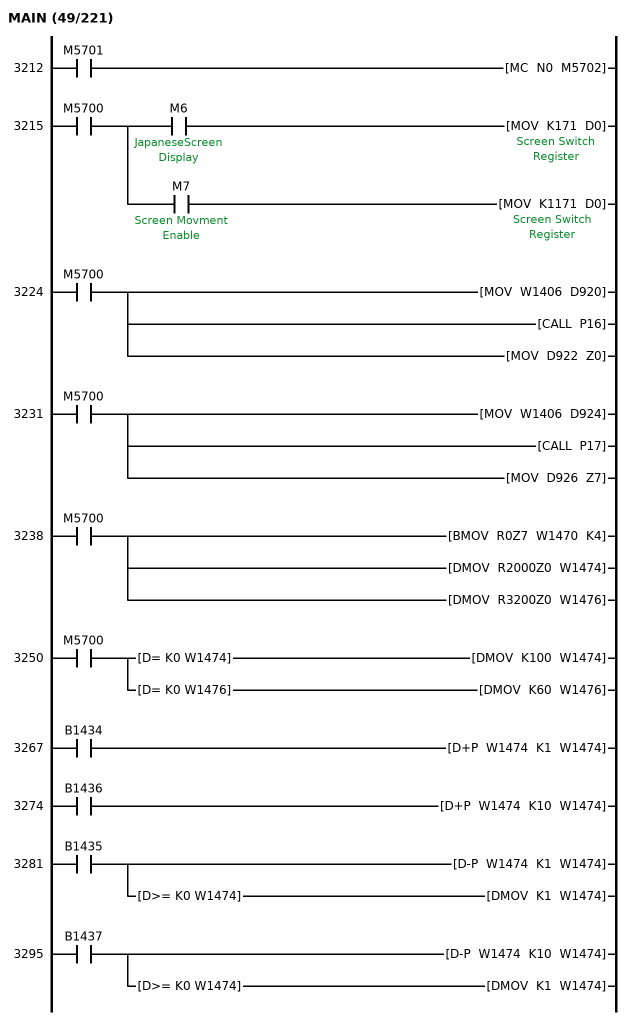
[picture p48: ladder of MAIN, rungs at steps 3212 to 3295]
3212  LD      M5701
      MC      N0 M5702
3215  LD      M5700
      MPS
      AND     M6  ; JapaneseScreen Display
      MOV     K171 D0
      MPP
      AND     M7  ; Screen Movment Enable
      MOV     K1171 D0
3224  LD      M5700
      MOV     W1406 D920
      CALL    P16
      MOV     D922 Z0
3231  LD      M5700
      MOV     W1406 D924
      CALL    P17
      MOV     D926 Z7
3238  LD      M5700
      BMOV    R0Z7 W1470 K4
      DMOV    R2000Z0 W1474
      DMOV    R3200Z0 W1476
3250  LD      M5700
      MPS
      ANDD=   K0 W1474
      DMOV    K100 W1474
      MPP
      ANDD=   K0 W1476
      DMOV    K60 W1476
3267  LD      B1434
      D+P     W1474 K1 W1474
3274  LD      B1436
      D+P     W1474 K10 W1474
3281  LD      B1435
      D-P     W1474 K1 W1474
      ANDD>=  K0 W1474
      DMOV    K1 W1474
3295  LD      B1437
      D-P     W1474 K10 W1474
      ANDD>=  K0 W1474
      DMOV    K1 W1474
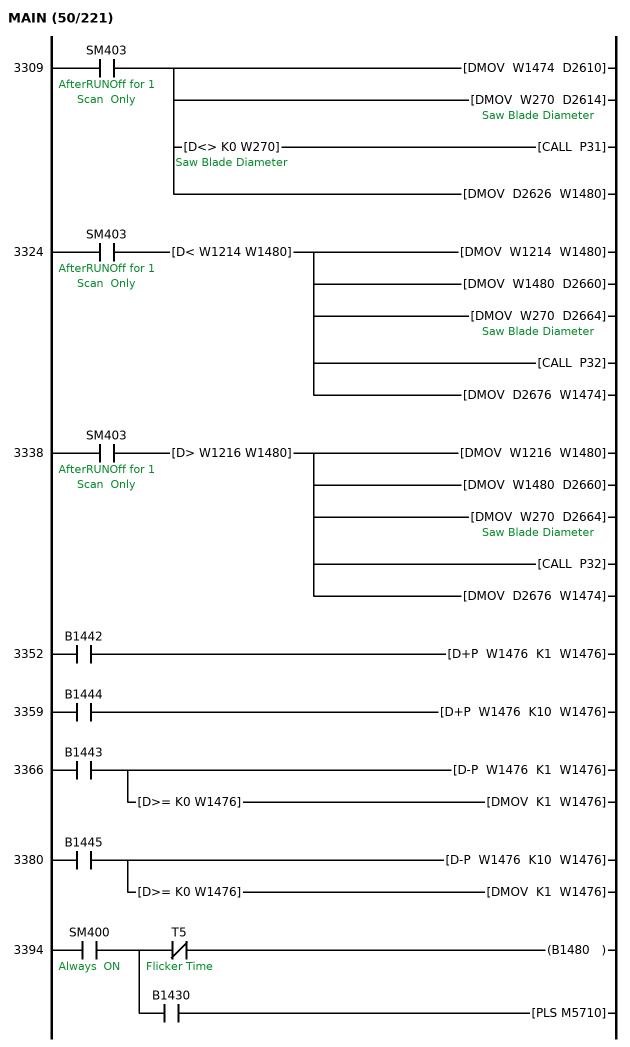
3309  LD      SM403  ; AfterRUNOff for 1 Scan  Only
      DMOV    W1474 D2610
      DMOV    W270 D2614
      MPS
      ANDD<>  K0 W270  ; Saw Blade Diameter
      CALL    P31
      MPP
      DMOV    D2626 W1480
3324  LD      SM403  ; AfterRUNOff for 1 Scan  Only
      ANDD<   W1214 W1480
      DMOV    W1214 W1480
      DMOV    W1480 D2660
      DMOV    W270 D2664
      CALL    P32
      DMOV    D2676 W1474
3338  LD      SM403  ; AfterRUNOff for 1 Scan  Only
      ANDD>   W1216 W1480
      DMOV    W1216 W1480
      DMOV    W1480 D2660
      DMOV    W270 D2664
      CALL    P32
      DMOV    D2676 W1474
3352  LD      B1442
      D+P     W1476 K1 W1476
3359  LD      B1444
      D+P     W1476 K10 W1476
3366  LD      B1443
      D-P     W1476 K1 W1476
      ANDD>=  K0 W1476
      DMOV    K1 W1476
3380  LD      B1445
      D-P     W1476 K10 W1476
      ANDD>=  K0 W1476
      DMOV    K1 W1476
3394  LD      SM400  ; Always  ON
      MPS
      ANI     T5  ; Flicker Time
      OUT     B1480
      MPP
      AND     B1430
      PLS     M5710
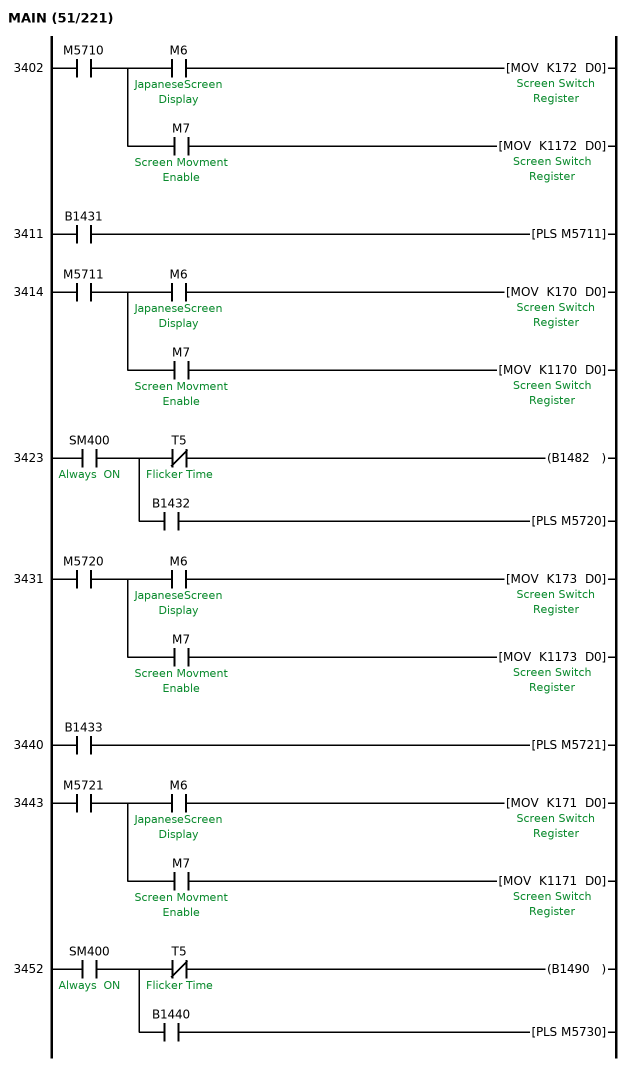
3402  LD      M5710
      MPS
      AND     M6  ; JapaneseScreen Display
      MOV     K172 D0
      MPP
      AND     M7  ; Screen Movment Enable
      MOV     K1172 D0
3411  LD      B1431
      PLS     M5711
3414  LD      M5711
      MPS
      AND     M6  ; JapaneseScreen Display
      MOV     K170 D0
      MPP
      AND     M7  ; Screen Movment Enable
      MOV     K1170 D0
3423  LD      SM400  ; Always  ON
      MPS
      ANI     T5  ; Flicker Time
      OUT     B1482
      MPP
      AND     B1432
      PLS     M5720
3431  LD      M5720
      MPS
      AND     M6  ; JapaneseScreen Display
      MOV     K173 D0
      MPP
      AND     M7  ; Screen Movment Enable
      MOV     K1173 D0
3440  LD      B1433
      PLS     M5721
3443  LD      M5721
      MPS
      AND     M6  ; JapaneseScreen Display
      MOV     K171 D0
      MPP
      AND     M7  ; Screen Movment Enable
      MOV     K1171 D0
3452  LD      SM400  ; Always  ON
      MPS
      ANI     T5  ; Flicker Time
      OUT     B1490
      MPP
      AND     B1440
      PLS     M5730
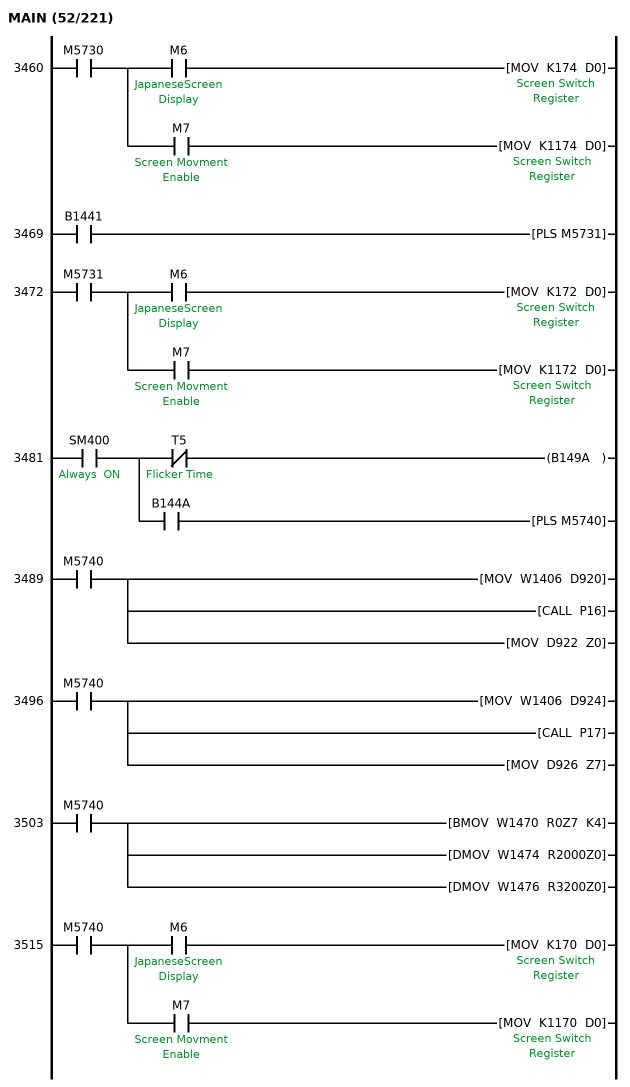
3460  LD      M5730
      MPS
      AND     M6  ; JapaneseScreen Display
      MOV     K174 D0
      MPP
      AND     M7  ; Screen Movment Enable
      MOV     K1174 D0
3469  LD      B1441
      PLS     M5731
3472  LD      M5731
      MPS
      AND     M6  ; JapaneseScreen Display
      MOV     K172 D0
      MPP
      AND     M7  ; Screen Movment Enable
      MOV     K1172 D0
3481  LD      SM400  ; Always  ON
      MPS
      ANI     T5  ; Flicker Time
      OUT     B149A
      MPP
      AND     B144A
      PLS     M5740
3489  LD      M5740
      MOV     W1406 D920
      CALL    P16
      MOV     D922 Z0
3496  LD      M5740
      MOV     W1406 D924
      CALL    P17
      MOV     D926 Z7
3503  LD      M5740
      BMOV    W1470 R0Z7 K4
      DMOV    W1474 R2000Z0
      DMOV    W1476 R3200Z0
3515  LD      M5740
      MPS
      AND     M6  ; JapaneseScreen Display
      MOV     K170 D0
      MPP
      AND     M7  ; Screen Movment Enable
      MOV     K1170 D0
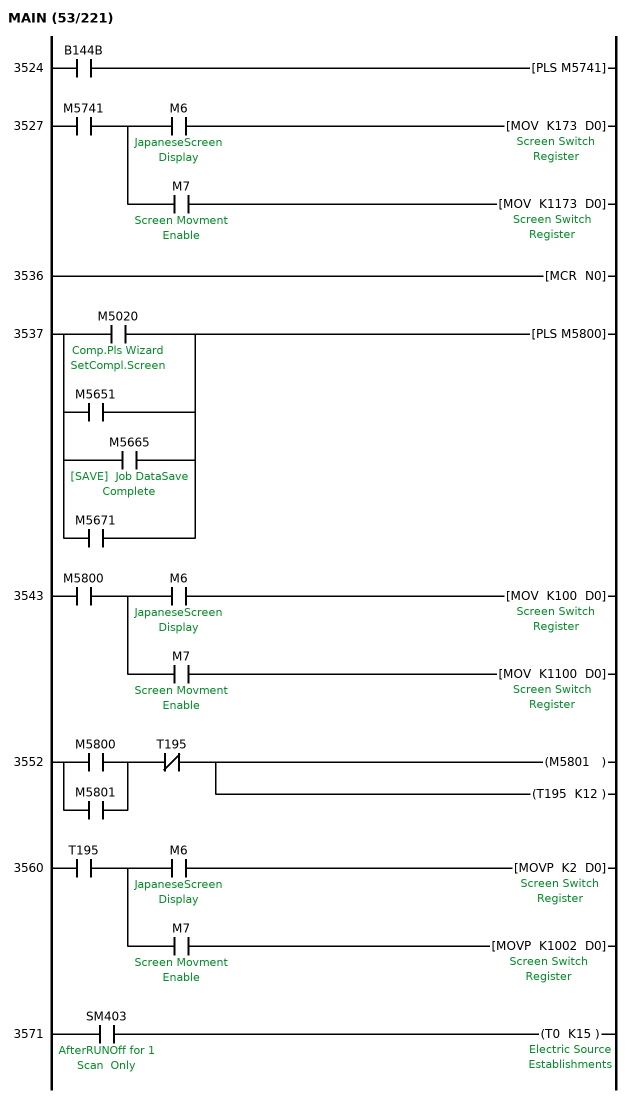
3524  LD      B144B
      PLS     M5741
3527  LD      M5741
      MPS
      AND     M6  ; JapaneseScreen Display
      MOV     K173 D0
      MPP
      AND     M7  ; Screen Movment Enable
      MOV     K1173 D0
3536  MCR     N0
3537  LD      M5020  ; Comp.Pls Wizard SetCompl.Screen
      OR      M5651
      OR      M5665  ; [SAVE]  Job DataSave Complete
      OR      M5671
      PLS     M5800
3543  LD      M5800
      MPS
      AND     M6  ; JapaneseScreen Display
      MOV     K100 D0
      MPP
      AND     M7  ; Screen Movment Enable
      MOV     K1100 D0
3552  LD      M5800
      OR      M5801
      ANI     T195
      OUT     M5801
      OUT     T195 K12
3560  LD      T195
      MPS
      AND     M6  ; JapaneseScreen Display
      MOVP    K2 D0
      MPP
      AND     M7  ; Screen Movment Enable
      MOVP    K1002 D0
3571  LD      SM403  ; AfterRUNOff for 1 Scan  Only
      OUT     T0 K15  ; Electric Source Establishments
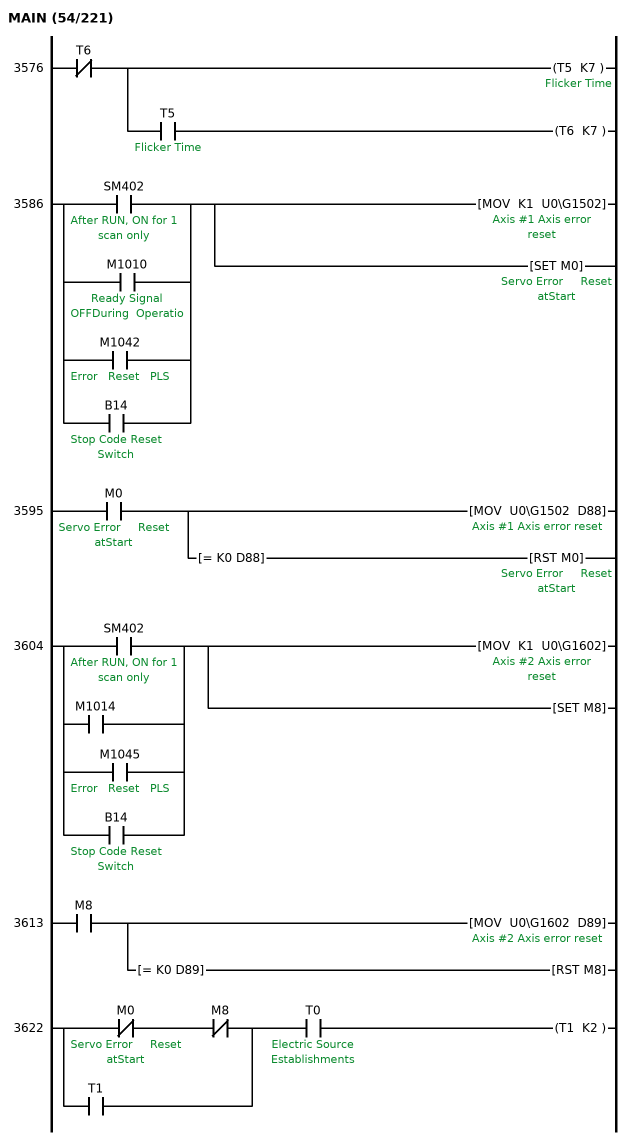
3576  LDI     T6
      OUT     T5 K7  ; Flicker Time
      AND     T5  ; Flicker Time
      OUT     T6 K7
3586  LD      SM402  ; After RUN, ON for 1 scan only
      OR      M1010  ; Ready Signal OFFDuring  Operatio
      OR      M1042  ; Error   Reset   PLS
      OR      B14  ; Stop Code Reset Switch
      MOV     K1 U0\G1502  ; Axis #1 Axis error reset
      SET     M0  ; Servo Error     Reset atStart
3595  LD      M0  ; Servo Error     Reset atStart
      MOV     U0\G1502 D88
      AND=    K0 D88
      RST     M0  ; Servo Error     Reset atStart
3604  LD      SM402  ; After RUN, ON for 1 scan only
      OR      M1014
      OR      M1045  ; Error   Reset   PLS
      OR      B14  ; Stop Code Reset Switch
      MOV     K1 U0\G1602  ; Axis #2 Axis error reset
      SET     M8
3613  LD      M8
      MOV     U0\G1602 D89
      AND=    K0 D89
      RST     M8
3622  LDI     M0  ; Servo Error     Reset atStart
      ANI     M8
      OR      T1
      AND     T0  ; Electric Source Establishments
      OUT     T1 K2
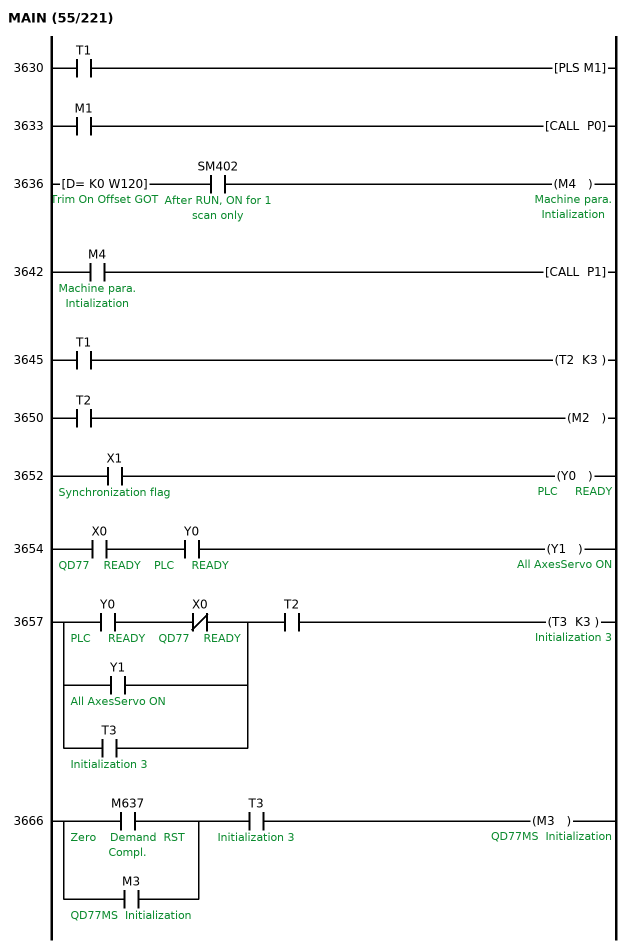
3630  LD      T1
      PLS     M1
3633  LD      M1
      CALL    P0
3636  LDD=    K0 W120  ; Trim On Offset GOT
      AND     SM402  ; After RUN, ON for 1 scan only
      OUT     M4  ; Machine para.   Intialization
3642  LD      M4  ; Machine para.   Intialization
      CALL    P1
3645  LD      T1
      OUT     T2 K3
3650  LD      T2
      OUT     M2
3652  LD      X1  ; Synchronization flag
      OUT     Y0  ; PLC     READY
3654  LD      X0  ; QD77    READY
      AND     Y0  ; PLC     READY
      OUT     Y1  ; All AxesServo ON
3657  LD      Y0  ; PLC     READY
      ANI     X0  ; QD77    READY
      OR      Y1  ; All AxesServo ON
      OR      T3  ; Initialization 3
      AND     T2
      OUT     T3 K3  ; Initialization 3
3666  LD      M637  ; Zero    Demand  RST     Compl.
      OR      M3  ; QD77MS  Initialization
      AND     T3  ; Initialization 3
      OUT     M3  ; QD77MS  Initialization
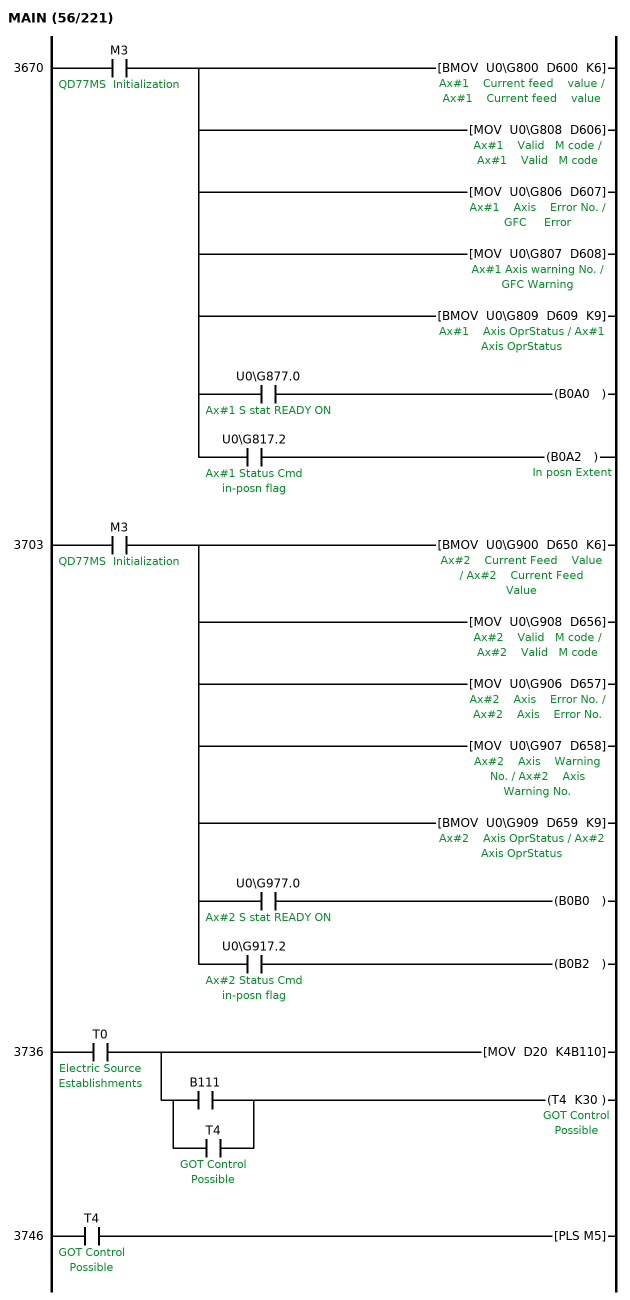
3670  LD      M3  ; QD77MS  Initialization
      BMOV    U0\G800 D600 K6  ; Ax#1    Current feed    value / Ax#1    Current feed    value
      MOV     U0\G808 D606  ; Ax#1    Valid   M code / Ax#1    Valid   M code
      MOV     U0\G806 D607  ; Ax#1    Axis    Error No. / GFC     Error
      MOV     U0\G807 D608  ; Ax#1 Axis warning No. / GFC Warning
      BMOV    U0\G809 D609 K9  ; Ax#1    Axis OprStatus / Ax#1    Axis OprStatus
      MPS
      AND     U0\G877.0  ; Ax#1 S stat READY ON
      OUT     B0A0
      MPP
      AND     U0\G817.2  ; Ax#1 Status Cmd in-posn flag
      OUT     B0A2  ; In posn Extent
3703  LD      M3  ; QD77MS  Initialization
      BMOV    U0\G900 D650 K6  ; Ax#2    Current Feed    Value / Ax#2    Current Feed    Value
      MOV     U0\G908 D656  ; Ax#2    Valid   M code / Ax#2    Valid   M code
      MOV     U0\G906 D657  ; Ax#2    Axis    Error No. / Ax#2    Axis    Error No.
      MOV     U0\G907 D658  ; Ax#2    Axis    Warning No. / Ax#2    Axis    Warning No.
      BMOV    U0\G909 D659 K9  ; Ax#2    Axis OprStatus / Ax#2    Axis OprStatus
      MPS
      AND     U0\G977.0  ; Ax#2 S stat READY ON
      OUT     B0B0
      MPP
      AND     U0\G917.2  ; Ax#2 Status Cmd in-posn flag
      OUT     B0B2
3736  LD      T0  ; Electric Source Establishments
      MOV     D20 K4B110
      LD      B111
      OR      T4  ; GOT Control     Possible
      ANB
      OUT     T4 K30  ; GOT Control     Possible
3746  LD      T4  ; GOT Control     Possible
      PLS     M5
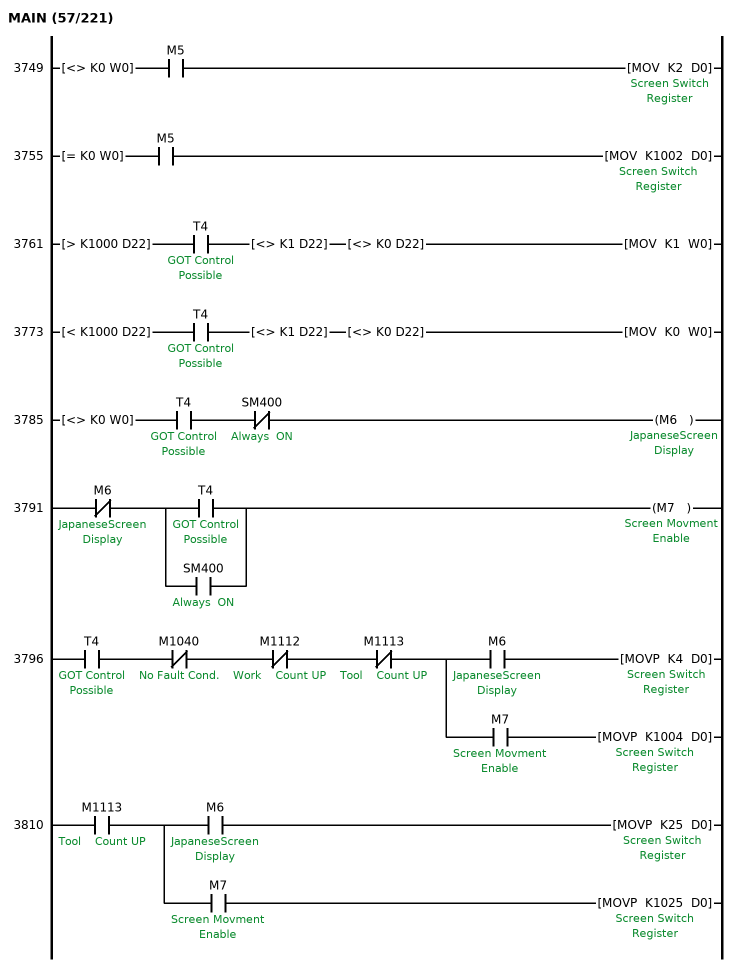
3749  LD<>    K0 W0
      AND     M5
      MOV     K2 D0
3755  LD=     K0 W0
      AND     M5
      MOV     K1002 D0
3761  LD>     K1000 D22
      AND     T4  ; GOT Control     Possible
      AND<>   K1 D22
      AND<>   K0 D22
      MOV     K1 W0
3773  LD<     K1000 D22
      AND     T4  ; GOT Control     Possible
      AND<>   K1 D22
      AND<>   K0 D22
      MOV     K0 W0
3785  LD<>    K0 W0
      AND     T4  ; GOT Control     Possible
      ANI     SM400  ; Always  ON
      OUT     M6  ; JapaneseScreen Display
3791  LDI     M6  ; JapaneseScreen Display
      LD      T4  ; GOT Control     Possible
      OR      SM400  ; Always  ON
      ANB
      OUT     M7  ; Screen Movment Enable
3796  LD      T4  ; GOT Control     Possible
      ANI     M1040  ; No Fault Cond.
      ANI     M1112  ; Work    Count UP
      ANI     M1113  ; Tool    Count UP
      MPS
      AND     M6  ; JapaneseScreen Display
      MOVP    K4 D0
      MPP
      AND     M7  ; Screen Movment Enable
      MOVP    K1004 D0
3810  LD      M1113  ; Tool    Count UP
      MPS
      AND     M6  ; JapaneseScreen Display
      MOVP    K25 D0
      MPP
      AND     M7  ; Screen Movment Enable
      MOVP    K1025 D0
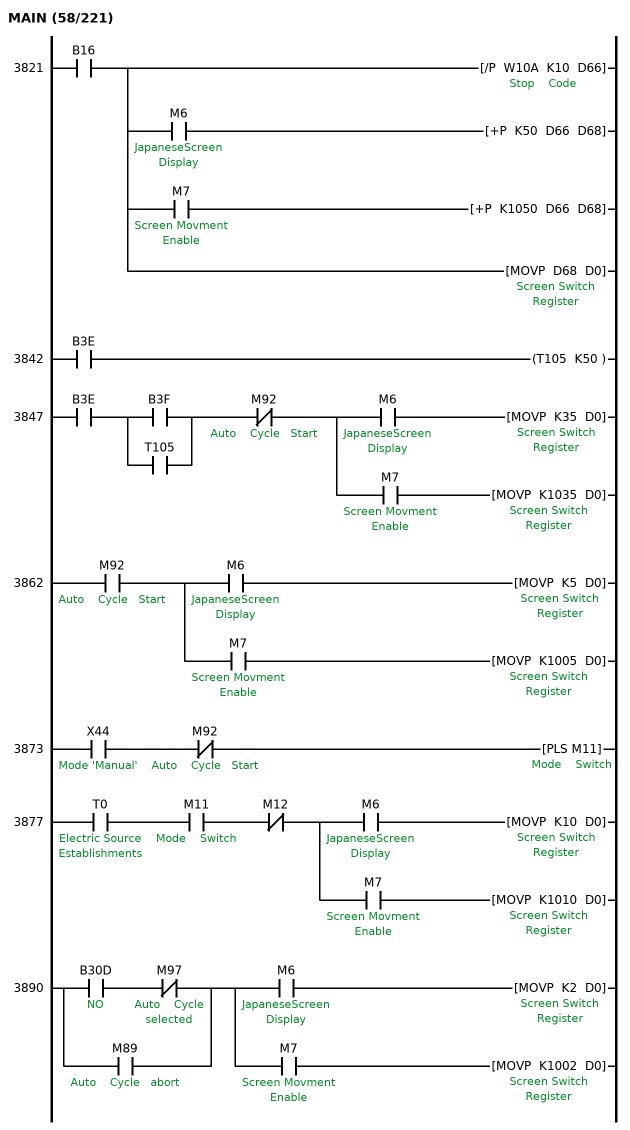
3821  LD      B16
      /P      W10A K10 D66  ; Stop    Code
      MPS
      AND     M6  ; JapaneseScreen Display
      +P      K50 D66 D68
      MRD
      AND     M7  ; Screen Movment Enable
      +P      K1050 D66 D68
      MPP
      MOVP    D68 D0
3842  LD      B3E
      OUT     T105 K50
3847  LD      B3E
      LD      B3F
      OR      T105
      ANB
      ANI     M92  ; Auto    Cycle   Start
      MPS
      AND     M6  ; JapaneseScreen Display
      MOVP    K35 D0
      MPP
      AND     M7  ; Screen Movment Enable
      MOVP    K1035 D0
3862  LD      M92  ; Auto    Cycle   Start
      MPS
      AND     M6  ; JapaneseScreen Display
      MOVP    K5 D0
      MPP
      AND     M7  ; Screen Movment Enable
      MOVP    K1005 D0
3873  LD      X44  ; Mode 'Manual'
      ANI     M92  ; Auto    Cycle   Start
      PLS     M11  ; Mode    Switch
3877  LD      T0  ; Electric Source Establishments
      AND     M11  ; Mode    Switch
      ANI     M12
      MPS
      AND     M6  ; JapaneseScreen Display
      MOVP    K10 D0
      MPP
      AND     M7  ; Screen Movment Enable
      MOVP    K1010 D0
3890  LD      B30D  ; NO
      ANI     M97  ; Auto    Cycle   selected
      OR      M89  ; Auto    Cycle   abort
      MPS
      AND     M6  ; JapaneseScreen Display
      MOVP    K2 D0
      MPP
      AND     M7  ; Screen Movment Enable
      MOVP    K1002 D0
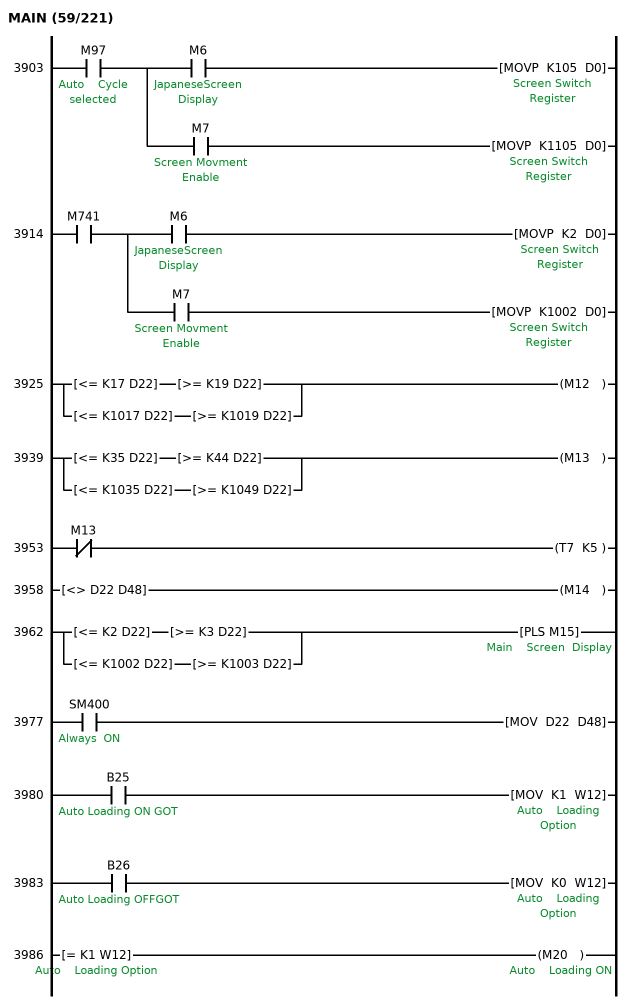
3903  LD      M97  ; Auto    Cycle   selected
      MPS
      AND     M6  ; JapaneseScreen Display
      MOVP    K105 D0
      MPP
      AND     M7  ; Screen Movment Enable
      MOVP    K1105 D0
3914  LD      M741
      MPS
      AND     M6  ; JapaneseScreen Display
      MOVP    K2 D0
      MPP
      AND     M7  ; Screen Movment Enable
      MOVP    K1002 D0
3925  LD<=    K17 D22
      AND>=   K19 D22
      LD<=    K1017 D22
      AND>=   K1019 D22
      ORB
      OUT     M12
3939  LD<=    K35 D22
      AND>=   K44 D22
      LD<=    K1035 D22
      AND>=   K1049 D22
      ORB
      OUT     M13
3953  LDI     M13
      OUT     T7 K5
3958  LD<>    D22 D48
      OUT     M14
3962  LD<=    K2 D22
      AND>=   K3 D22
      LD<=    K1002 D22
      AND>=   K1003 D22
      ORB
      PLS     M15  ; Main    Screen  Display
3977  LD      SM400  ; Always  ON
      MOV     D22 D48
3980  LD      B25  ; Auto Loading ON GOT
      MOV     K1 W12  ; Auto    Loading Option
3983  LD      B26  ; Auto Loading OFFGOT
      MOV     K0 W12
3986  LD=     K1 W12  ; Auto    Loading Option
      OUT     M20  ; Auto    Loading ON
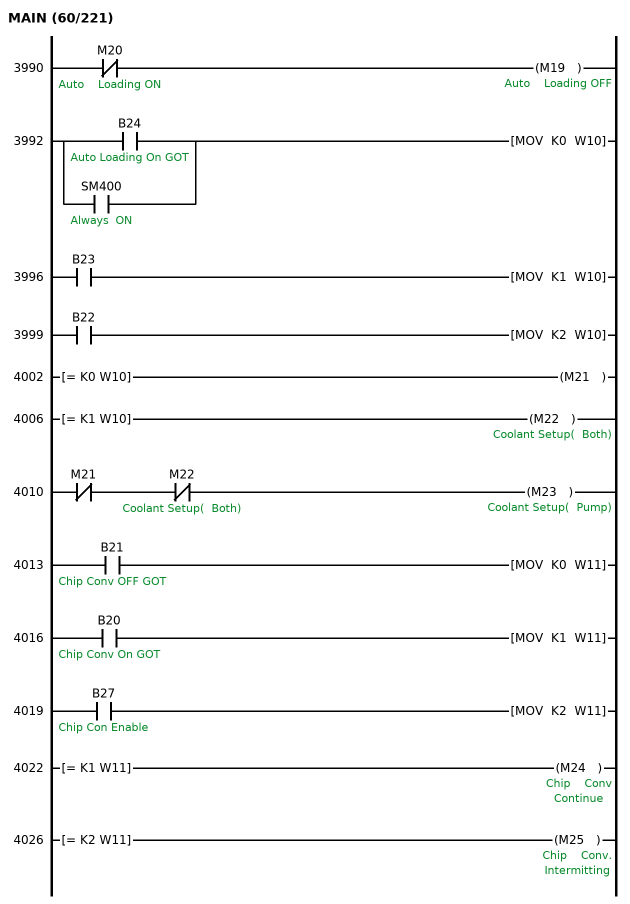
3990  LDI     M20  ; Auto    Loading ON
      OUT     M19  ; Auto    Loading OFF
3992  LD      B24  ; Auto Loading On GOT
      OR      SM400  ; Always  ON
      MOV     K0 W10
3996  LD      B23
      MOV     K1 W10
3999  LD      B22
      MOV     K2 W10
4002  LD=     K0 W10
      OUT     M21
4006  LD=     K1 W10
      OUT     M22  ; Coolant Setup(  Both)
4010  LDI     M21
      ANI     M22  ; Coolant Setup(  Both)
      OUT     M23  ; Coolant Setup(  Pump)
4013  LD      B21  ; Chip Conv OFF GOT
      MOV     K0 W11
4016  LD      B20  ; Chip Conv On GOT
      MOV     K1 W11
4019  LD      B27  ; Chip Con Enable
      MOV     K2 W11
4022  LD=     K1 W11
      OUT     M24  ; Chip    Conv    Continue
4026  LD=     K2 W11
      OUT     M25  ; Chip    Conv.   Intermitting
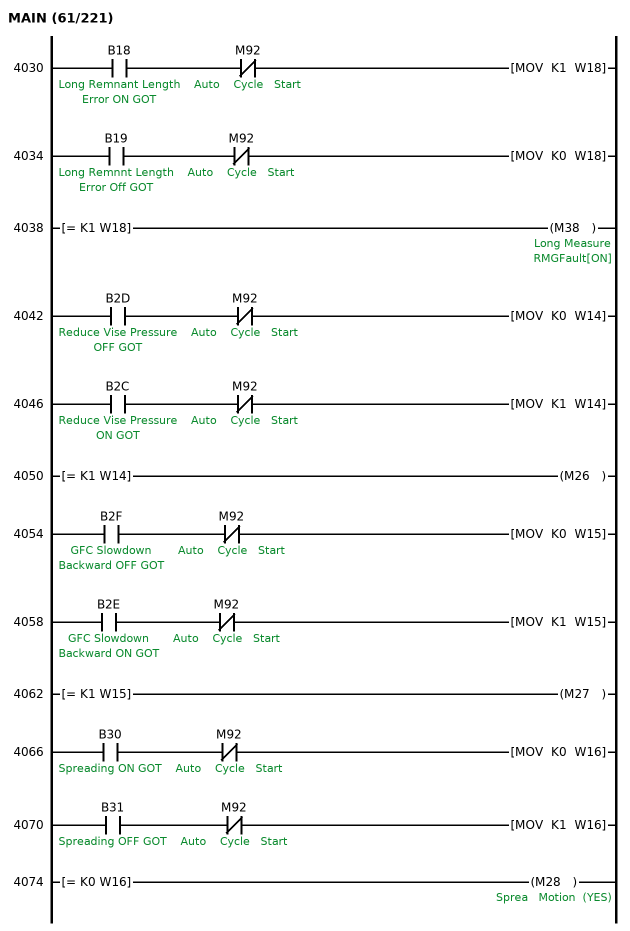
4030  LD      B18  ; Long Remnant Length Error ON GOT
      ANI     M92  ; Auto    Cycle   Start
      MOV     K1 W18
4034  LD      B19  ; Long Remnnt Length Error Off GOT
      ANI     M92  ; Auto    Cycle   Start
      MOV     K0 W18
4038  LD=     K1 W18
      OUT     M38  ; Long Measure RMGFault[ON]
4042  LD      B2D  ; Reduce Vise Pressure OFF GOT
      ANI     M92  ; Auto    Cycle   Start
      MOV     K0 W14
4046  LD      B2C  ; Reduce Vise Pressure ON GOT
      ANI     M92  ; Auto    Cycle   Start
      MOV     K1 W14
4050  LD=     K1 W14
      OUT     M26
4054  LD      B2F  ; GFC Slowdown Backward OFF GOT
      ANI     M92  ; Auto    Cycle   Start
      MOV     K0 W15
4058  LD      B2E  ; GFC Slowdown Backward ON GOT
      ANI     M92  ; Auto    Cycle   Start
      MOV     K1 W15
4062  LD=     K1 W15
      OUT     M27
4066  LD      B30  ; Spreading ON GOT
      ANI     M92  ; Auto    Cycle   Start
      MOV     K0 W16
4070  LD      B31  ; Spreading OFF GOT
      ANI     M92  ; Auto    Cycle   Start
      MOV     K1 W16
4074  LD=     K0 W16
      OUT     M28  ; Sprea   Motion  (YES)
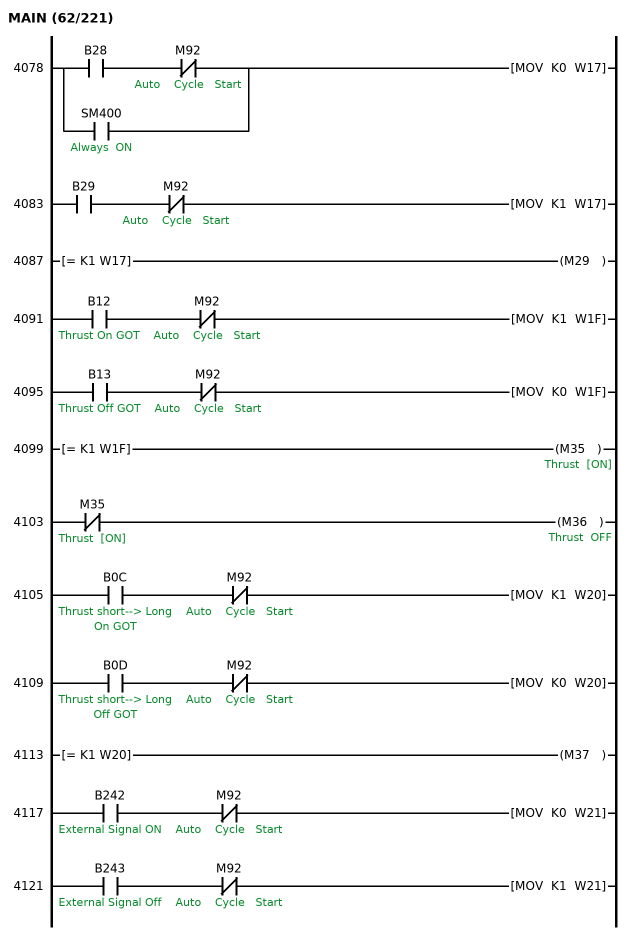
4078  LD      B28
      ANI     M92  ; Auto    Cycle   Start
      OR      SM400  ; Always  ON
      MOV     K0 W17
4083  LD      B29
      ANI     M92  ; Auto    Cycle   Start
      MOV     K1 W17
4087  LD=     K1 W17
      OUT     M29
4091  LD      B12  ; Thrust On GOT
      ANI     M92  ; Auto    Cycle   Start
      MOV     K1 W1F
4095  LD      B13  ; Thrust Off GOT
      ANI     M92  ; Auto    Cycle   Start
      MOV     K0 W1F
4099  LD=     K1 W1F
      OUT     M35  ; Thrust  [ON]
4103  LDI     M35  ; Thrust  [ON]
      OUT     M36  ; Thrust  OFF
4105  LD      B0C  ; Thrust short--> Long On GOT
      ANI     M92  ; Auto    Cycle   Start
      MOV     K1 W20
4109  LD      B0D  ; Thrust short--> Long Off GOT
      ANI     M92  ; Auto    Cycle   Start
      MOV     K0 W20
4113  LD=     K1 W20
      OUT     M37
4117  LD      B242  ; External Signal ON
      ANI     M92  ; Auto    Cycle   Start
      MOV     K0 W21
4121  LD      B243  ; External Signal Off
      ANI     M92  ; Auto    Cycle   Start
      MOV     K1 W21
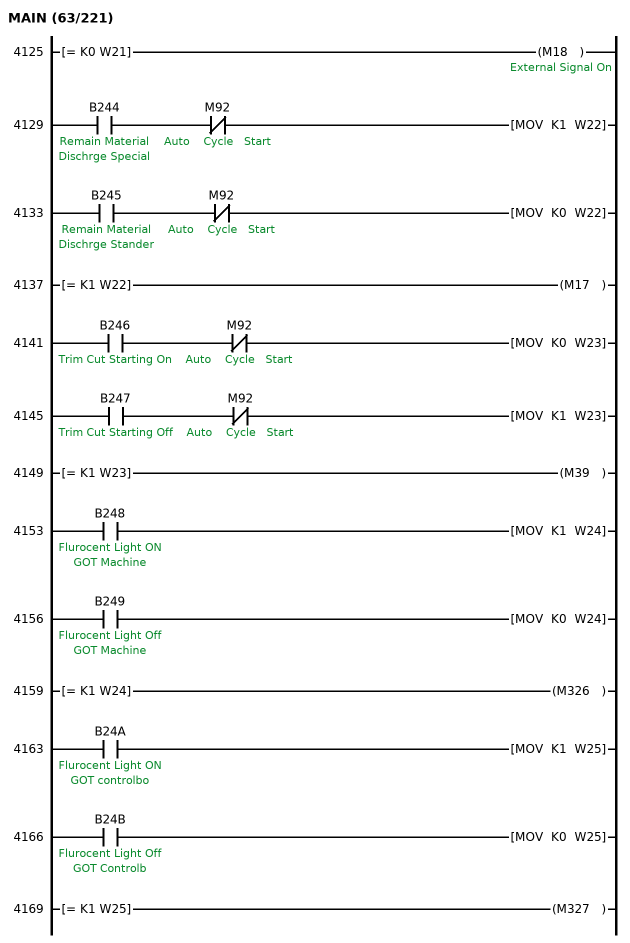
4125  LD=     K0 W21
      OUT     M18  ; External Signal On
4129  LD      B244  ; Remain Material Dischrge Special
      ANI     M92  ; Auto    Cycle   Start
      MOV     K1 W22
4133  LD      B245  ; Remain Material Dischrge Stander
      ANI     M92  ; Auto    Cycle   Start
      MOV     K0 W22
4137  LD=     K1 W22
      OUT     M17
4141  LD      B246  ; Trim Cut Starting On
      ANI     M92  ; Auto    Cycle   Start
      MOV     K0 W23
4145  LD      B247  ; Trim Cut Starting Off
      ANI     M92  ; Auto    Cycle   Start
      MOV     K1 W23
4149  LD=     K1 W23
      OUT     M39
4153  LD      B248  ; Flurocent Light ON GOT Machine
      MOV     K1 W24
4156  LD      B249  ; Flurocent Light Off GOT Machine
      MOV     K0 W24
4159  LD=     K1 W24
      OUT     M326
4163  LD      B24A  ; Flurocent Light ON GOT controlbo
      MOV     K1 W25
4166  LD      B24B  ; Flurocent Light Off GOT Controlb
      MOV     K0 W25
4169  LD=     K1 W25
      OUT     M327
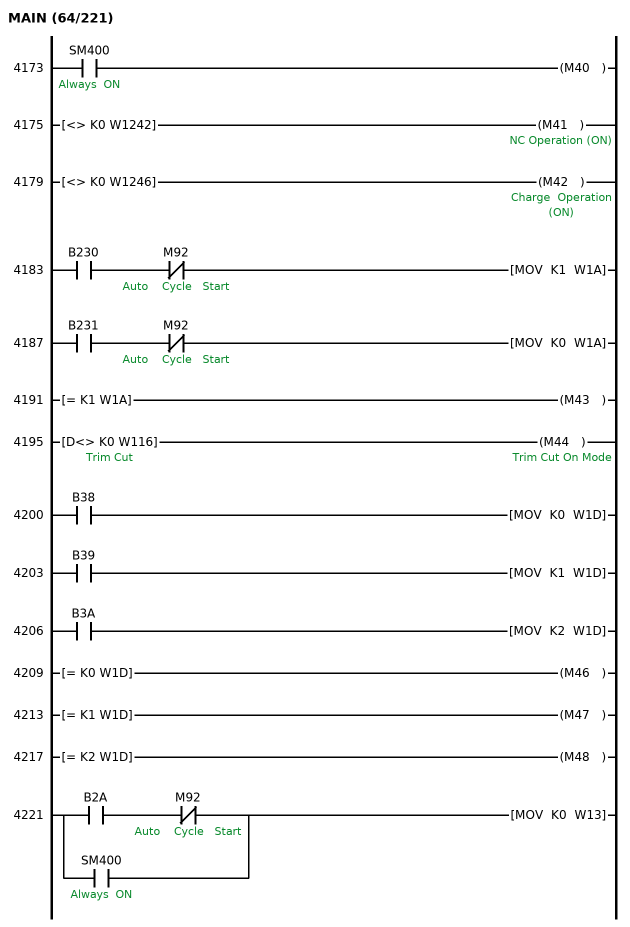
4173  LD      SM400  ; Always  ON
      OUT     M40
4175  LD<>    K0 W1242
      OUT     M41  ; NC Operation (ON)
4179  LD<>    K0 W1246
      OUT     M42  ; Charge  Operation (ON)
4183  LD      B230
      ANI     M92  ; Auto    Cycle   Start
      MOV     K1 W1A
4187  LD      B231
      ANI     M92  ; Auto    Cycle   Start
      MOV     K0 W1A
4191  LD=     K1 W1A
      OUT     M43
4195  LDD<>   K0 W116  ; Trim Cut
      OUT     M44  ; Trim Cut On Mode
4200  LD      B38
      MOV     K0 W1D
4203  LD      B39
      MOV     K1 W1D
4206  LD      B3A
      MOV     K2 W1D
4209  LD=     K0 W1D
      OUT     M46
4213  LD=     K1 W1D
      OUT     M47
4217  LD=     K2 W1D
      OUT     M48
4221  LD      B2A
      ANI     M92  ; Auto    Cycle   Start
      OR      SM400  ; Always  ON
      MOV     K0 W13
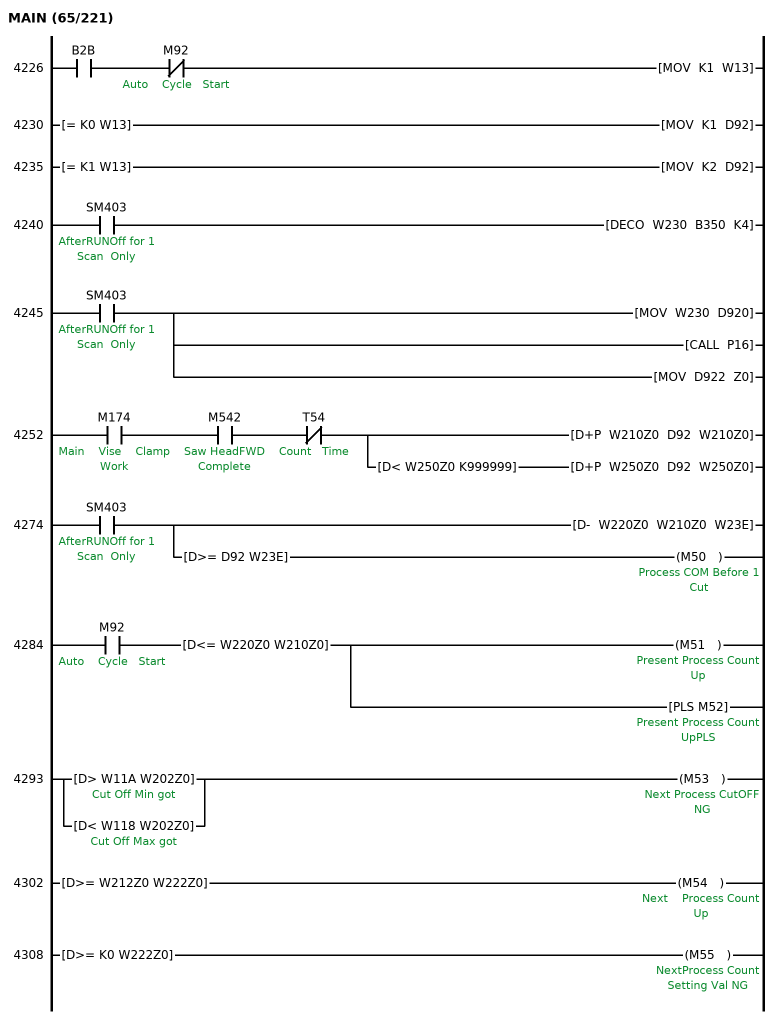
4226  LD      B2B
      ANI     M92  ; Auto    Cycle   Start
      MOV     K1 W13
4230  LD=     K0 W13
      MOV     K1 D92
4235  LD=     K1 W13
      MOV     K2 D92
4240  LD      SM403  ; AfterRUNOff for 1 Scan  Only
      DECO    W230 B350 K4
4245  LD      SM403  ; AfterRUNOff for 1 Scan  Only
      MOV     W230 D920
      CALL    P16
      MOV     D922 Z0
4252  LD      M174  ; Main    Vise    Clamp   Work
      AND     M542  ; Saw HeadFWD     Complete
      ANI     T54  ; Count   Time
      D+P     W210Z0 D92 W210Z0
      ANDD<   W250Z0 K999999
      D+P     W250Z0 D92 W250Z0
4274  LD      SM403  ; AfterRUNOff for 1 Scan  Only
      D-      W220Z0 W210Z0 W23E
      ANDD>=  D92 W23E
      OUT     M50  ; Process COM Before 1 Cut
4284  LD      M92  ; Auto    Cycle   Start
      ANDD<=  W220Z0 W210Z0
      OUT     M51  ; Present Process Count Up
      PLS     M52  ; Present Process Count UpPLS
4293  LDD>    W11A W202Z0  ; Cut Off Min got
      ORD<    W118 W202Z0  ; Cut Off Max got
      OUT     M53  ; Next Process CutOFF NG
4302  LDD>=   W212Z0 W222Z0
      OUT     M54  ; Next    Process Count Up
4308  LDD>=   K0 W222Z0
      OUT     M55  ; NextProcess Count Setting Val NG
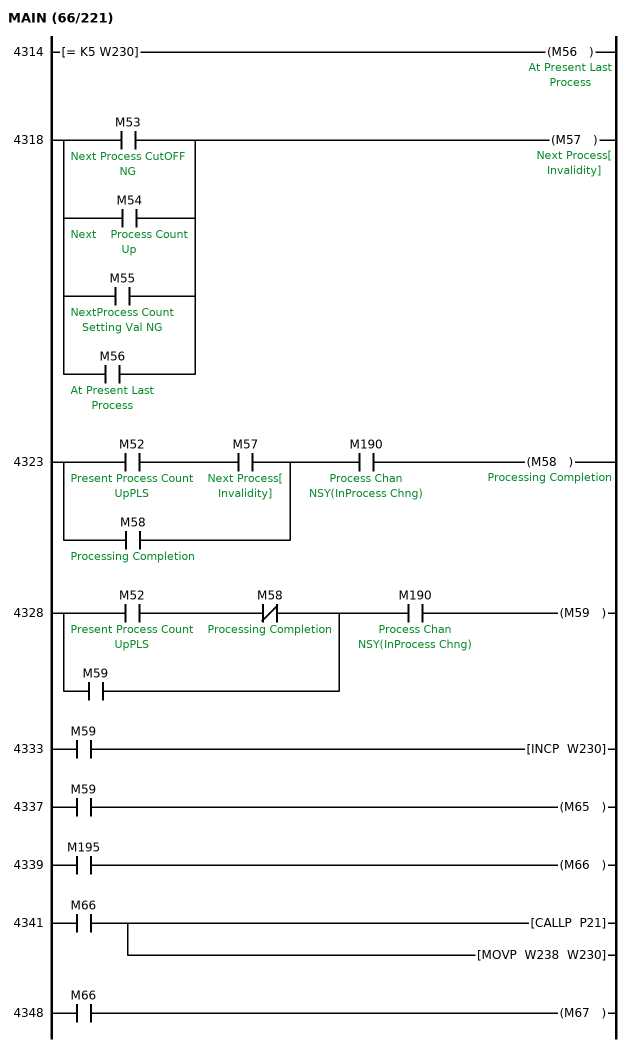
4314  LD=     K5 W230
      OUT     M56  ; At Present Last Process
4318  LD      M53  ; Next Process CutOFF NG
      OR      M54  ; Next    Process Count Up
      OR      M55  ; NextProcess Count Setting Val NG
      OR      M56  ; At Present Last Process
      OUT     M57  ; Next Process[Invalidity]
4323  LD      M52  ; Present Process Count UpPLS
      AND     M57  ; Next Process[Invalidity]
      OR      M58  ; Processing Completion
      AND     M190  ; Process Chan NSY(InProcess Chng)
      OUT     M58  ; Processing Completion
4328  LD      M52  ; Present Process Count UpPLS
      ANI     M58  ; Processing Completion
      OR      M59
      AND     M190  ; Process Chan NSY(InProcess Chng)
      OUT     M59
4333  LD      M59
      INCP    W230
4337  LD      M59
      OUT     M65
4339  LD      M195
      OUT     M66
4341  LD      M66
      CALLP   P21
      MOVP    W238 W230
4348  LD      M66
      OUT     M67
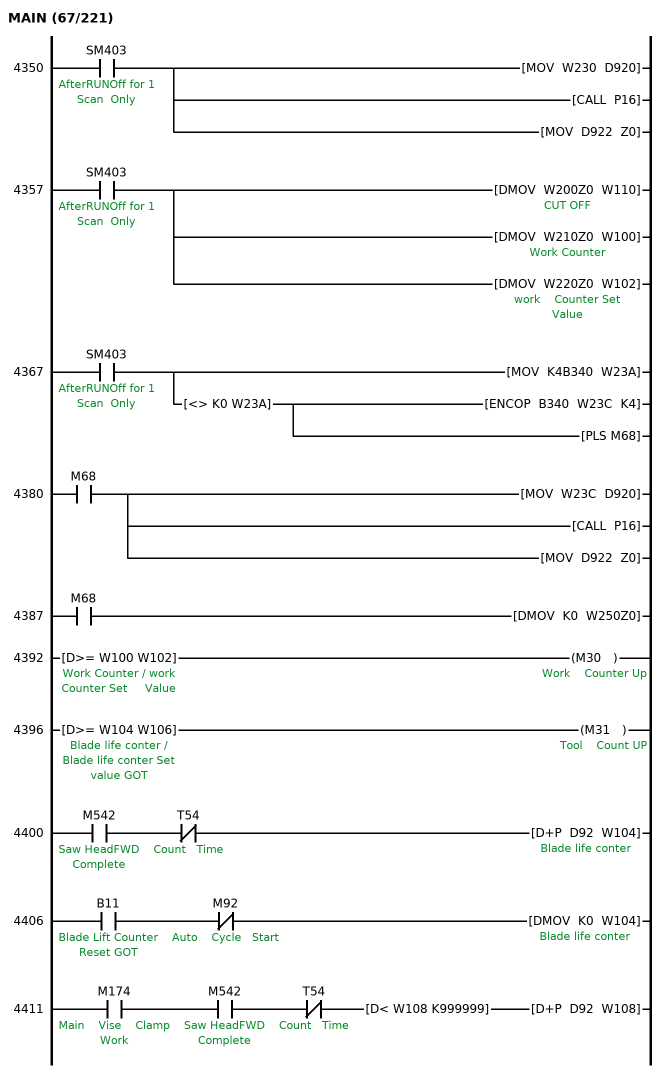
4350  LD      SM403  ; AfterRUNOff for 1 Scan  Only
      MOV     W230 D920
      CALL    P16
      MOV     D922 Z0
4357  LD      SM403  ; AfterRUNOff for 1 Scan  Only
      DMOV    W200Z0 W110  ; CUT OFF
      DMOV    W210Z0 W100  ; Work Counter
      DMOV    W220Z0 W102  ; work    Counter Set     Value
4367  LD      SM403  ; AfterRUNOff for 1 Scan  Only
      MOV     K4B340 W23A
      AND<>   K0 W23A
      ENCOP   B340 W23C K4
      PLS     M68
4380  LD      M68
      MOV     W23C D920
      CALL    P16
      MOV     D922 Z0
4387  LD      M68
      DMOV    K0 W250Z0
4392  LDD>=   W100 W102  ; Work Counter / work    Counter Set     Value
      OUT     M30  ; Work    Counter Up
4396  LDD>=   W104 W106  ; Blade life conter / Blade life conter Set value GOT
      OUT     M31  ; Tool    Count UP
4400  LD      M542  ; Saw HeadFWD     Complete
      ANI     T54  ; Count   Time
      D+P     D92 W104
4406  LD      B11  ; Blade Lift Counter Reset GOT
      ANI     M92  ; Auto    Cycle   Start
      DMOV    K0 W104
4411  LD      M174  ; Main    Vise    Clamp   Work
      AND     M542  ; Saw HeadFWD     Complete
      ANI     T54  ; Count   Time
      ANDD<   W108 K999999
      D+P     D92 W108
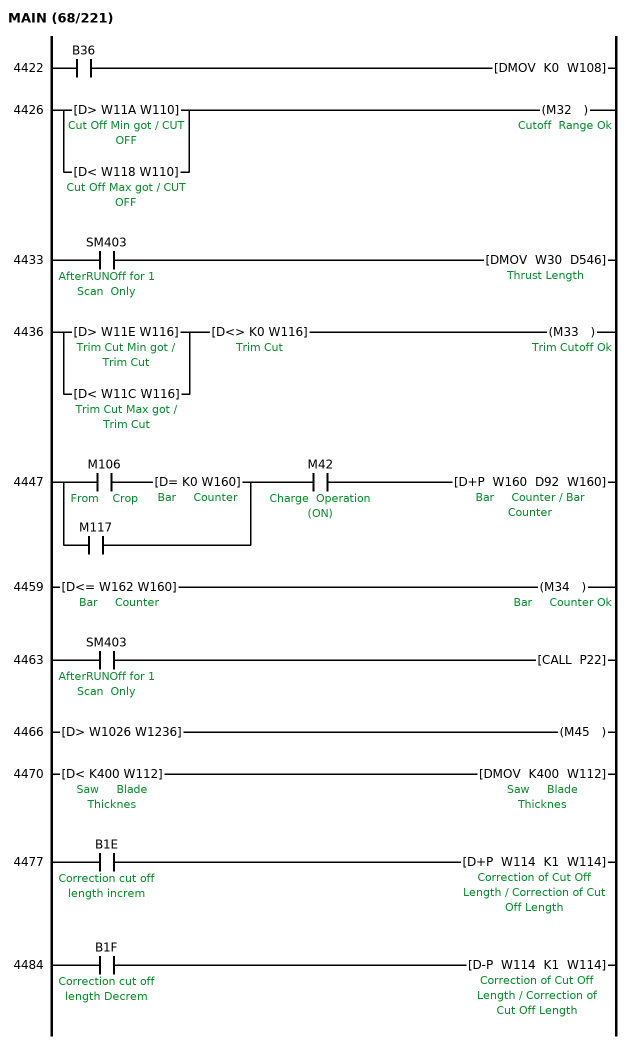
4422  LD      B36
      DMOV    K0 W108
4426  LDD>    W11A W110  ; Cut Off Min got / CUT OFF
      ORD<    W118 W110  ; Cut Off Max got / CUT OFF
      OUT     M32  ; Cutoff  Range Ok
4433  LD      SM403  ; AfterRUNOff for 1 Scan  Only
      DMOV    W30 D546  ; Thrust Length
4436  LDD>    W11E W116  ; Trim Cut Min got / Trim Cut
      ORD<    W11C W116  ; Trim Cut Max got / Trim Cut
      ANDD<>  K0 W116  ; Trim Cut
      OUT     M33  ; Trim Cutoff Ok
4447  LD      M106  ; From    Crop
      ANDD=   K0 W160  ; Bar     Counter
      OR      M117
      AND     M42  ; Charge  Operation (ON)
      D+P     W160 D92 W160
4459  LDD<=   W162 W160  ; Bar     Counter
      OUT     M34  ; Bar     Counter Ok
4463  LD      SM403  ; AfterRUNOff for 1 Scan  Only
      CALL    P22
4466  LDD>    W1026 W1236
      OUT     M45
4470  LDD<    K400 W112  ; Saw     Blade   Thicknes
      DMOV    K400 W112
4477  LD      B1E  ; Correction cut off length increm
      D+P     W114 K1 W114  ; Correction of Cut Off Length
4484  LD      B1F  ; Correction cut off length Decrem
      D-P     W114 K1 W114
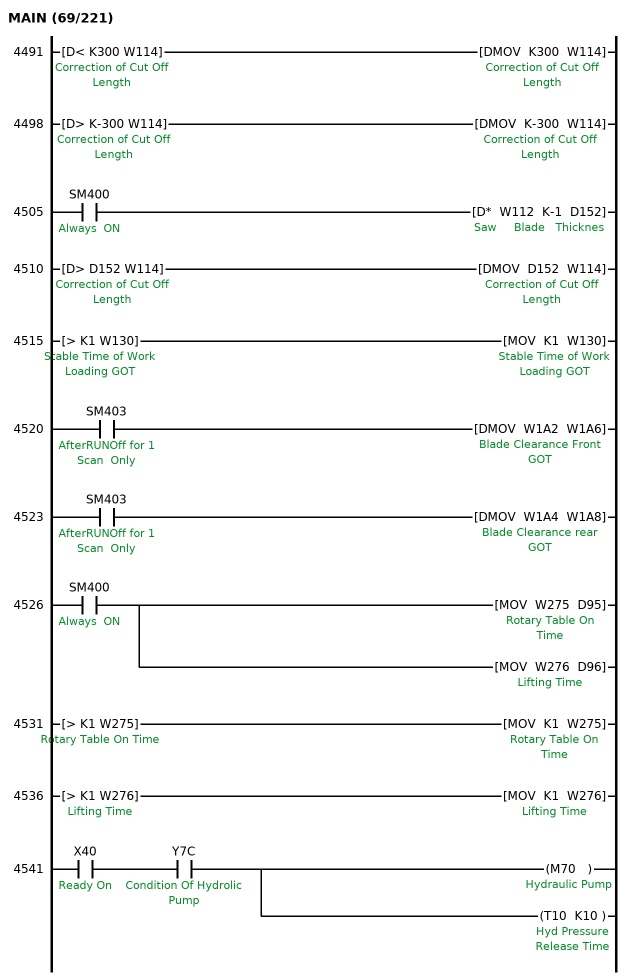
4491  LDD<    K300 W114  ; Correction of Cut Off Length
      DMOV    K300 W114
4498  LDD>    K-300 W114  ; Correction of Cut Off Length
      DMOV    K-300 W114
4505  LD      SM400  ; Always  ON
      D*      W112 K-1 D152
4510  LDD>    D152 W114  ; Correction of Cut Off Length
      DMOV    D152 W114
4515  LD>     K1 W130  ; Stable Time of Work Loading GOT
      MOV     K1 W130
4520  LD      SM403  ; AfterRUNOff for 1 Scan  Only
      DMOV    W1A2 W1A6  ; Blade Clearance Front GOT
4523  LD      SM403  ; AfterRUNOff for 1 Scan  Only
      DMOV    W1A4 W1A8  ; Blade Clearance rear GOT
4526  LD      SM400  ; Always  ON
      MOV     W275 D95  ; Rotary Table On Time
      MOV     W276 D96  ; Lifting Time
4531  LD>     K1 W275  ; Rotary Table On Time
      MOV     K1 W275
4536  LD>     K1 W276  ; Lifting Time
      MOV     K1 W276
4541  LD      X40  ; Ready On
      AND     Y7C  ; Condition Of Hydrolic Pump
      OUT     M70  ; Hydraulic Pump
      OUT     T10 K10  ; Hyd Pressure    Release Time
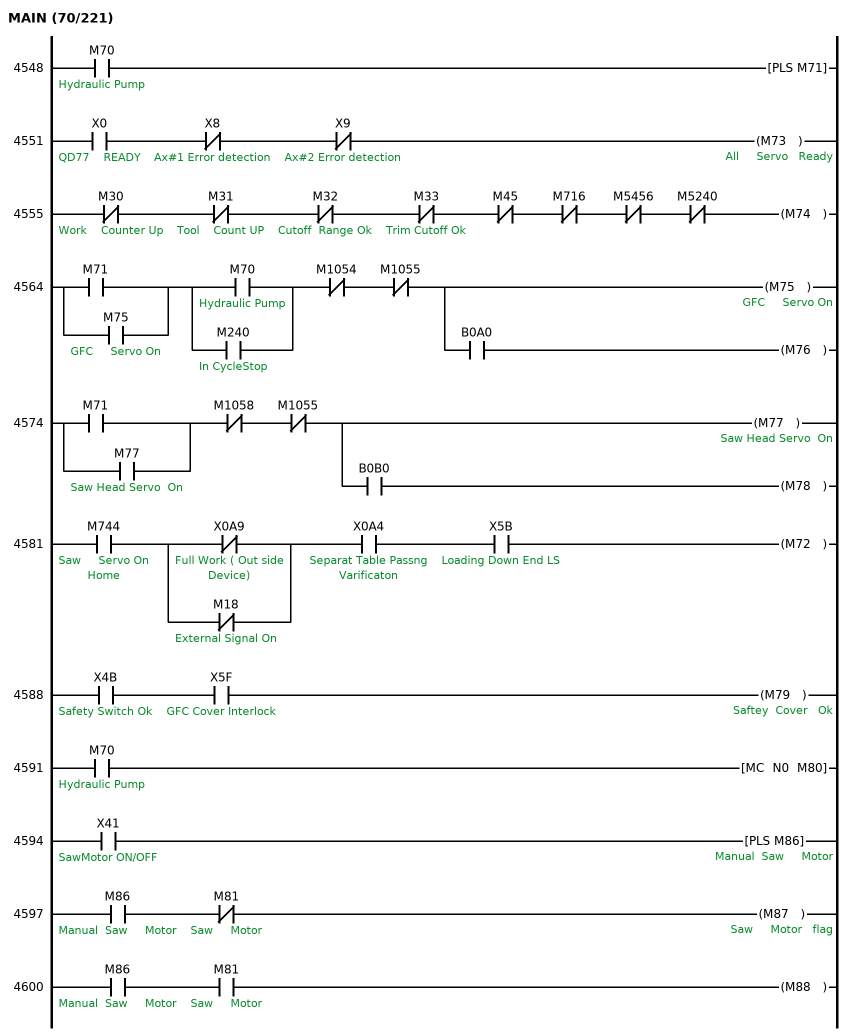
4548  LD      M70  ; Hydraulic Pump
      PLS     M71
4551  LD      X0  ; QD77    READY
      ANI     X8  ; Ax#1 Error detection
      ANI     X9  ; Ax#2 Error detection
      OUT     M73  ; All     Servo   Ready
4555  LDI     M30  ; Work    Counter Up
      ANI     M31  ; Tool    Count UP
      ANI     M32  ; Cutoff  Range Ok
      ANI     M33  ; Trim Cutoff Ok
      ANI     M45
      ANI     M716
      ANI     M5456
      ANI     M5240
      OUT     M74
4564  LD      M71
      OR      M75  ; GFC     Servo On
      LD      M70  ; Hydraulic Pump
      OR      M240  ; In CycleStop
      ANB
      ANI     M1054
      ANI     M1055
      OUT     M75  ; GFC     Servo On
      AND     B0A0
      OUT     M76
4574  LD      M71
      OR      M77  ; Saw Head Servo  On
      ANI     M1058
      ANI     M1055
      OUT     M77  ; Saw Head Servo  On
      AND     B0B0
      OUT     M78
4581  LD      M744  ; Saw     Servo On Home
      LDI     X0A9  ; Full Work ( Out side Device)
      ORI     M18  ; External Signal On
      ANB
      AND     X0A4  ; Separat Table Passng Varificaton
      AND     X5B  ; Loading Down End LS
      OUT     M72
4588  LD      X4B  ; Safety Switch Ok
      AND     X5F  ; GFC Cover Interlock
      OUT     M79  ; Saftey  Cover   Ok
4591  LD      M70  ; Hydraulic Pump
      MC      N0 M80
4594  LD      X41  ; SawMotor ON/OFF
      PLS     M86  ; Manual  Saw     Motor
4597  LD      M86  ; Manual  Saw     Motor
      ANI     M81  ; Saw     Motor
      OUT     M87  ; Saw     Motor   flag
4600  LD      M86  ; Manual  Saw     Motor
      AND     M81  ; Saw     Motor
      OUT     M88
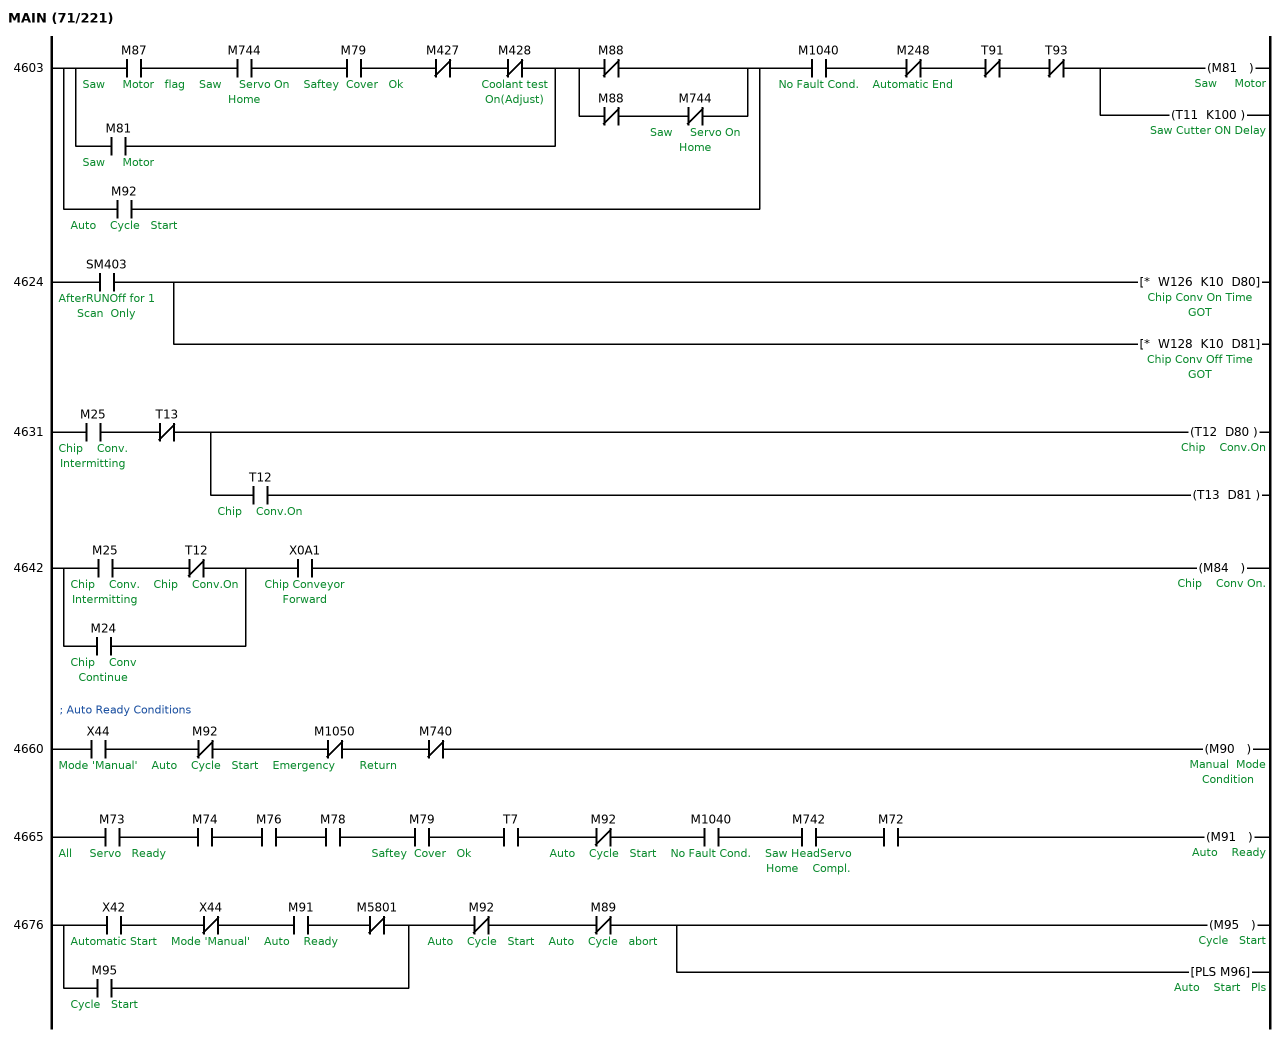
4603  LD      M87  ; Saw     Motor   flag
      AND     M744  ; Saw     Servo On Home
      AND     M79  ; Saftey  Cover   Ok
      ANI     M427
      ANI     M428  ; Coolant test On(Adjust)
      OR      M81  ; Saw     Motor
      LDI     M88
      LDI     M88
      ANI     M744  ; Saw     Servo On Home
      ORB
      ANB
      OR      M92  ; Auto    Cycle   Start
      AND     M1040  ; No Fault Cond.
      ANI     M248  ; Automatic End
      ANI     T91
      ANI     T93
      OUT     M81  ; Saw     Motor
      OUT     T11 K100  ; Saw Cutter ON Delay
4624  LD      SM403  ; AfterRUNOff for 1 Scan  Only
      *       W126 K10 D80  ; Chip Conv On Time GOT
      *       W128 K10 D81  ; Chip Conv Off Time GOT
4631  LD      M25  ; Chip    Conv.   Intermitting
      ANI     T13
      OUT     T12 D80  ; Chip    Conv.On
      AND     T12  ; Chip    Conv.On
      OUT     T13 D81
4642  LD      M25  ; Chip    Conv.   Intermitting
      ANI     T12  ; Chip    Conv.On
      OR      M24  ; Chip    Conv    Continue
      AND     X0A1  ; Chip Conveyor Forward
      OUT     M84  ; Chip    Conv On.
; Auto Ready Conditions
4660  LD      X44  ; Mode 'Manual'
      ANI     M92  ; Auto    Cycle   Start
      ANI     M1050  ; Emergency       Return
      ANI     M740
      OUT     M90  ; Manual  Mode    Condition
4665  LD      M73  ; All     Servo   Ready
      AND     M74
      AND     M76
      AND     M78
      AND     M79  ; Saftey  Cover   Ok
      AND     T7
      ANI     M92  ; Auto    Cycle   Start
      AND     M1040  ; No Fault Cond.
      AND     M742  ; Saw HeadServo   Home    Compl.
      AND     M72
      OUT     M91  ; Auto    Ready
4676  LD      X42  ; Automatic Start
      ANI     X44  ; Mode 'Manual'
      AND     M91  ; Auto    Ready
      ANI     M5801
      OR      M95  ; Cycle   Start
      ANI     M92  ; Auto    Cycle   Start
      ANI     M89  ; Auto    Cycle   abort
      OUT     M95  ; Cycle   Start
      PLS     M96  ; Auto    Start   Pls
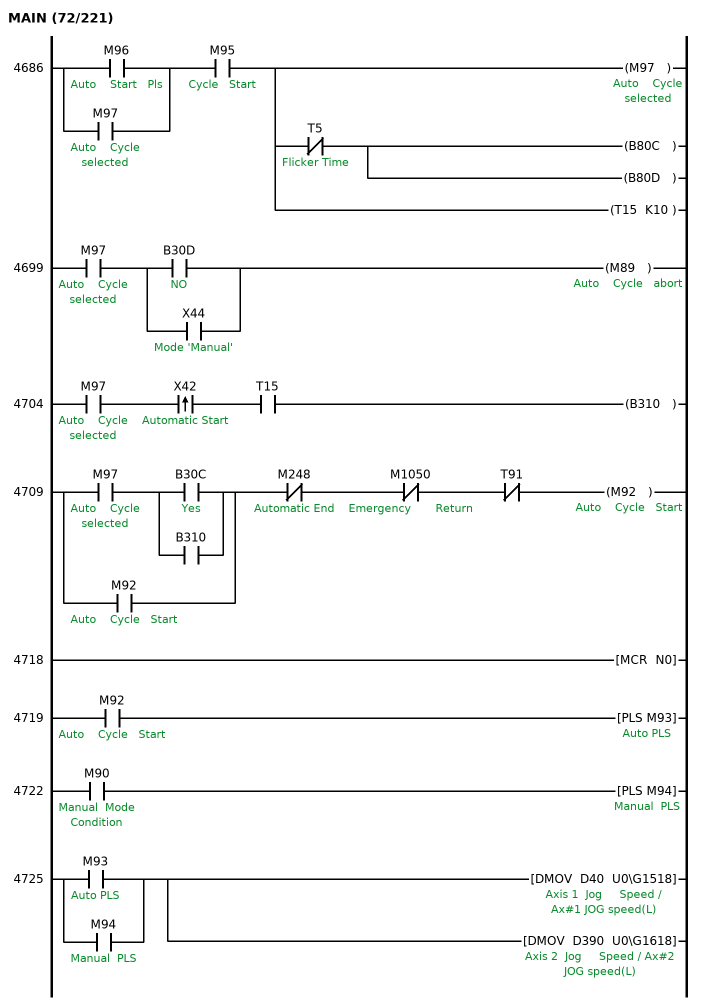
4686  LD      M96  ; Auto    Start   Pls
      OR      M97  ; Auto    Cycle   selected
      AND     M95  ; Cycle   Start
      OUT     M97  ; Auto    Cycle   selected
      MPS
      ANI     T5  ; Flicker Time
      OUT     B80C
      OUT     B80D
      MPP
      OUT     T15 K10
4699  LD      M97  ; Auto    Cycle   selected
      LD      B30D  ; NO
      OR      X44  ; Mode 'Manual'
      ANB
      OUT     M89  ; Auto    Cycle   abort
4704  LD      M97  ; Auto    Cycle   selected
      ANDP    X42  ; Automatic Start
      AND     T15
      OUT     B310
4709  LD      M97  ; Auto    Cycle   selected
      LD      B30C  ; Yes
      OR      B310
      ANB
      OR      M92  ; Auto    Cycle   Start
      ANI     M248  ; Automatic End
      ANI     M1050  ; Emergency       Return
      ANI     T91
      OUT     M92  ; Auto    Cycle   Start
4718  MCR     N0
4719  LD      M92  ; Auto    Cycle   Start
      PLS     M93  ; Auto PLS
4722  LD      M90  ; Manual  Mode    Condition
      PLS     M94  ; Manual  PLS
4725  LD      M93  ; Auto PLS
      OR      M94  ; Manual  PLS
      DMOV    D40 U0\G1518  ; Axis 1  Jog     Speed / Ax#1 JOG speed(L)
      DMOV    D390 U0\G1618  ; Axis 2  Jog     Speed / Ax#2 JOG speed(L)
